FUNCTION_BLOCK FB_Function EXTENDS FB_Component
VAR_INPUT
END_VAR
VAR_OUTPUT
END_VAR
VAR
END_VAR

END_FUNCTION_BLOCK

(* stored: Version 1.1.0.1
   POU FB_Function: Id {a9649e04-0f5a-0a2d-2ecf-08f61b920136}, SpecialFunc None *)
